(* CODESYS project Raspihats.library
   Description: Library for raspihats.com boards.
   Version: 1.0.0.0
   Title: Raspihats
   Author: Florin Costa
   DocFormat: reStructuredText
   Placeholder: Raspihats
   LanguageModelAttribute: qualified-access-only
   DefaultNamespace: Raspihats
   Company: Dabatop Industries SRL

Project tree, tasks and I/O mapping:
  libraries: Memory, 3.5.7.0 (3S - Smart Software Solutions GmbH); Raspberry Pi Peripherals, 3.5.13.0 (3S - Smart Software Solutions GmbH)
  I2CHAT/
    Globals/
      global variables I2CHAT_GVL
      data type I2CHAT_Command
      data type I2CHAT_ErrorCode
    Frame/
      function block I2CHAT_EncodeFrame [ST]
      function block I2CHAT_DecodeFrame [ST]
    Boards/
      function block I2CHAT_DI6acDQ6rly [ST]: AfterReadInputs, BeforeWriteOutputs
      function block I2CHAT_DI16ac [ST]: AfterReadInputs
      function block I2CHAT_DQ10rly [ST]: BeforeWriteOutputs
    I/O/
      function block I2CHAT_Transfer [ST]
      function block I2CHAT_DQ_Write [ST]
      function block I2CHAT_DI_Read [ST]
*)

// I2CHAT/Globals/I2CHAT_Command
{attribute 'qualified_only'}
{attribute 'strict'}
TYPE I2CHAT_Command :
(
    GET_BOARD_NAME                      := 16#10, 
    GET_FIRMWARE_VERSION                := 16#11, 
    GET_STATUS_WORD                     := 16#12, 
    RESET                               := 16#13,
 
    CWDT_SET_PERIOD                     := 16#14, 
    CWDT_GET_PERIOD                     := 16#15, 
    IRQ_GET_REG                         := 16#16, 
    IRQ_SET_REG                         := 16#17,  
 
    DI_GET_VALUE                        := 16#20, 
    DI_GET_CHANNEL_STATE                := 16#21, 
    DI_GET_COUNTER                      := 16#22, 
    DI_RESET_COUNTER                    := 16#23, 
    DI_RESET_ALL_COUNTERS               := 16#24, 
    DI_GET_COUNTERS_STATUS              := 16#25, 
    DI_GET_ENCODER                      := 16#26, 
    DI_RESET_ENCODER                    := 16#27, 
    DI_RESET_ALL_ENCODERS               := 16#28, 
    DI_GET_ENCODERS_STATUS              := 16#29, 
 
    DO_SET_POWER_ON_VALUE               := 16#30, 
    DO_GET_POWER_ON_VALUE               := 16#31, 
    DO_SET_SAFETY_VALUE                 := 16#32, 
    DO_GET_SAFETY_VALUE                 := 16#33, 
    DO_SET_VALUE                        := 16#34, 
    DO_GET_VALUE                        := 16#35, 
    DO_SET_CHANNEL_STATE                := 16#36, 
    DO_GET_CHANNEL_STATE                := 16#37
) USINT;
END_TYPE

// I2CHAT/Globals/I2CHAT_ErrorCode
{attribute 'qualified_only'}
{attribute 'strict'}
TYPE I2CHAT_ErrorCode :
(
	NO_ERROR := 0,
	I2C_WRITE_INCOMPLETE := 1,
	I2C_READ_INCOMPLETE := 2,
	BUFFER_OVERFLOW := 3,
	CRC_FAIL := 4,
	BAD_RESPONSE := 5
) UINT;
END_TYPE

// I2CHAT/Globals/I2CHAT_GVL
{attribute 'qualified_only'}
VAR_GLOBAL CONSTANT
	gc_uiFrameMinSize : UINT := 4; // 1(Id) + 1(Cmd) + 0(Payload) + 2(CRC16)
	gc_uiCrc16Size : UINT := 2;
END_VAR
VAR_GLOBAL
	g_usiFrameId : USINT := 0;
END_VAR

// I2CHAT/Boards/I2CHAT_DI6acDQ6rly
FUNCTION_BLOCK I2CHAT_DI6acDQ6rly EXTENDS i2c
VAR_INPUT
	udiDQValue : UDINT;
END_VAR
VAR_OUTPUT
	udiDIValue : UDINT;
	eErrorCode : I2CHAT_ErrorCode;
END_VAR
VAR
END_VAR

SUPER^();

CASE _iState OF
0:	
	IF SUPER^.init() THEN
		_iState := 10;
	END_IF	
	
END_CASE

METHOD AfterReadInputs : INT
VAR
	DI_Read : I2CHAT_DI_Read;
END_VAR
SUPER^.AfterReadInputs();

IF _iState = 10 THEN
	DI_Read(
		pI2CSlave := THIS
	);
	
	udiDIValue := DI_Read.udiValue;
	eErrorCode := DI_Read.eErrorCode;
END_IF
END_METHOD

METHOD BeforeWriteOutputs : INT
VAR
	DQ_Write : I2CHAT_DQ_Write;
	DI_Read: INT;
END_VAR
SUPER^.BeforeWriteOutputs();

IF _iState = 10 THEN
	DQ_Write(
		pI2CSlave := THIS, 
		udiValue := udiDQValue
	);
	
	eErrorCode := DQ_Write.eErrorCode;
END_IF
END_METHOD

END_FUNCTION_BLOCK

// I2CHAT/I/O/I2CHAT_DI_Read
FUNCTION_BLOCK I2CHAT_DI_Read
VAR_INPUT
	pI2CSlave : POINTER TO RasPi.i2c;
END_VAR
VAR_OUTPUT
	udiValue : UDINT;
	eErrorCode : I2CHAT_ErrorCode;
END_VAR
VAR
	ausiResponseData : ARRAY [0..3] OF USINT;
	Transfer : I2CHAT_Transfer;
END_VAR

Transfer(
	pI2CSlave := pI2CSlave,
	usiRequestCmd := I2CHAT_Command.DI_GET_VALUE,
	pusiRequestData := 0,
	uiRequestDataSize := 0,
	pusiResponseData := ADR(ausiResponseData),
	uiResponseDataSize := 4
);

IF Transfer.eErrorCode <> I2CHAT_ErrorCode.NO_ERROR THEN
	eErrorCode := Transfer.eErrorCode;
	RETURN;
END_IF

udiValue := ausiResponseData[0];
udiValue := udiValue + SHL(USINT_TO_UDINT(ausiResponseData[1]), 8);
udiValue := udiValue + SHL(USINT_TO_UDINT(ausiResponseData[2]), 16);
udiValue := udiValue + SHL(USINT_TO_UDINT(ausiResponseData[3]), 24);

END_FUNCTION_BLOCK

// I2CHAT/I/O/I2CHAT_Transfer
FUNCTION_BLOCK I2CHAT_Transfer
VAR_INPUT
	pI2CSlave : POINTER TO RasPi.i2c;
	usiRequestCmd : USINT;
	pusiRequestData : POINTER TO USINT;
	uiRequestDataSize : UINT;
	pusiResponseData : POINTER TO USINT;
	uiResponseDataSize : UINT;
END_VAR
VAR_OUTPUT
	eErrorCode : I2CHAT_ErrorCode;
END_VAR
VAR
	ausiBuffer : ARRAY [0..255] OF USINT;
	EncodeFrame : I2CHAT_EncodeFrame;
	DecodeFrame : I2CHAT_DecodeFrame;
	uiByteCnt : DINT;
END_VAR

eErrorCode := I2CHAT_ErrorCode.NO_ERROR;

I2CHAT_GVL.g_usiFrameId := (I2CHAT_GVL.g_usiFrameId + 1) AND 16#FF;

EncodeFrame(
	usiId := I2CHAT_GVL.g_usiFrameId,
	usiCmd := usiRequestCmd,
	pusiData := pusiRequestData,
	uiDataSize := uiRequestDataSize,
	pusiBuffer := ADR(ausiBuffer),
	uiBufferSize := SIZEOF(ausiBuffer)
);

IF EncodeFrame.eErrorCode <> I2CHAT_ErrorCode.NO_ERROR THEN
	eErrorCode := EncodeFrame.eErrorCode;
	RETURN;
END_IF

// Write I2C-HAT request
uiByteCnt := pI2CSlave^.write(ADR(ausiBuffer), EncodeFrame.uiEncodeSize);
IF uiByteCnt <> EncodeFrame.uiEncodeSize THEN
	eErrorCode := I2CHAT_ErrorCode.I2C_WRITE_INCOMPLETE;
	RETURN;
END_IF

// Read I2C-HAT response
uiByteCnt:= pI2CSlave^.read(ADR(ausiBuffer), I2CHAT_GVL.gc_uiFrameMinSize + uiResponseDataSize);
IF uiByteCnt <> (I2CHAT_GVL.gc_uiFrameMinSize + uiResponseDataSize) THEN
	eErrorCode := I2CHAT_ErrorCode.I2C_READ_INCOMPLETE;
	RETURN;
END_IF

DecodeFrame(
	pusiBuffer := ADR(ausiBuffer),
	uiBufferSize := I2CHAT_GVL.gc_uiFrameMinSize + uiResponseDataSize,
	pusiData := pusiResponseData,
	uiDataSize := uiResponseDataSize
);

IF DecodeFrame.eErrorCode <> I2CHAT_ErrorCode.NO_ERROR THEN
	eErrorCode := DecodeFrame.eErrorCode;
	RETURN;
END_IF

IF DecodeFrame.usiId <> EncodeFrame.usiId OR DecodeFrame.usiCmd <> EncodeFrame.usiCmd THEN
	eErrorCode := I2CHAT_ErrorCode.BAD_RESPONSE;
END_IF

END_FUNCTION_BLOCK

// I2CHAT/Frame/I2CHAT_EncodeFrame
FUNCTION_BLOCK I2CHAT_EncodeFrame
VAR_INPUT
	// input frame
	usiId : USINT;
	usiCmd : USINT;
	pusiData : POINTER TO USINT;
	uiDataSize : UINT;
	// encode buffer
	pusiBuffer : POINTER TO USINT;
	uiBufferSize : UINT;
END_VAR
VAR_OUTPUT
	uiEncodeSize : UINT;
	eErrorCode : I2CHAT_ErrorCode;
END_VAR
VAR
	uiEncodeIndex : UINT;
	uiIndex : UINT;
	uiCrc16 : UINT;
END_VAR

IF (I2CHAT_GVL.gc_uiFrameMinSize + uiDataSize) <= uiBufferSize THEN
	uiEncodeIndex := 0;
	
	pusiBuffer[uiEncodeIndex] := usiId;
	uiEncodeIndex := uiEncodeIndex + 1;
    
	pusiBuffer[uiEncodeIndex] := usiCmd;
	uiEncodeIndex := uiEncodeIndex + 1;

	IF uiDataSize > 0 THEN
		FOR uiIndex := 0 TO uiDataSize - 1 DO
			pusiBuffer[uiEncodeIndex] := pusiData[uiIndex];
			uiEncodeIndex := uiEncodeIndex + 1;		
		END_FOR
	END_IF

	uiCrc16 := MEM.CRC16_Modbus(pMemoryBlock := pusiBuffer, uiLength := uiEncodeIndex);

	pusiBuffer[uiEncodeIndex] := UINT_TO_USINT(uiCrc16);
	uiEncodeIndex := uiEncodeIndex + 1;
	
	pusiBuffer[uiEncodeIndex] := UINT_TO_USINT(SHR(uiCrc16, 8));
	uiEncodeIndex := uiEncodeIndex + 1;	
	
	uiEncodeSize := uiEncodeIndex;
	eErrorCode := I2CHAT_ErrorCode.NO_ERROR;
ELSE 
	uiEncodeSize := 0;	// Nothing Encoded
	eErrorCode := I2CHAT_ErrorCode.BUFFER_OVERFLOW;
END_IF

END_FUNCTION_BLOCK

// I2CHAT/Frame/I2CHAT_DecodeFrame
FUNCTION_BLOCK I2CHAT_DecodeFrame
VAR_INPUT
	// decode buffer
	pusiBuffer : POINTER TO USINT;
	uiBufferSize : UINT;
	// frame payload buffer
	pusiData : POINTER TO USINT;
	uiDataSize : UINT;
END_VAR
VAR_OUTPUT
	usiId : USINT;
	usiCmd : USINT;
	uiDecodeSize : UINT;
	eErrorCode : I2CHAT_ErrorCode;
END_VAR
VAR
	uiDecodeIndex : UINT;
	uiIndex : UINT;
	uiCrc16 : UINT;
END_VAR

IF uiBufferSize >= I2CHAT_GVL.gc_uiFrameMinSize AND uiDataSize >= (uiBufferSize - I2CHAT_GVL.gc_uiFrameMinSize) THEN
	uiDecodeIndex := 0;
	
	usiId := pusiBuffer[uiDecodeIndex]; 
	uiDecodeIndex := uiDecodeIndex + 1;
    
	usiCmd := pusiBuffer[uiDecodeIndex]; 
	uiDecodeIndex := uiDecodeIndex + 1;

	uiDataSize := uiBufferSize - I2CHAT_GVL.gc_uiFrameMinSize;
	IF uiDataSize > 0 THEN
		FOR uiIndex := 0 TO uiDataSize - 1 DO
			pusiData[uiIndex] := pusiBuffer[uiDecodeIndex];
			uiDecodeIndex := uiDecodeIndex + 1;	
		END_FOR
	END_IF

	uiCrc16 := USINT_TO_UINT(pusiBuffer[uiDecodeIndex]); 
	uiDecodeIndex := uiDecodeIndex + 1;
	
	uiCrc16 := uiCrc16 + SHL(USINT_TO_UINT(pusiBuffer[uiDecodeIndex]), 8); 
	uiDecodeIndex := uiDecodeIndex + 1;
	
	IF MEM.CRC16_Modbus(pMemoryBlock := pusiBuffer, uiLength := uiDecodeIndex - I2CHAT_GVL.gc_uiCrc16Size) = uiCrc16 THEN
		uiDecodeSize := uiDecodeIndex;
		eErrorCode := I2CHAT_ErrorCode.NO_ERROR;
	ELSE
		uiDecodeSize := 0;	
		eErrorCode := I2CHAT_ErrorCode.CRC_FAIL;
	END_IF
ELSE 
	uiDecodeSize := 0;
	eErrorCode := I2CHAT_ErrorCode.BUFFER_OVERFLOW;
END_IF

END_FUNCTION_BLOCK

// I2CHAT/I/O/I2CHAT_DQ_Write
FUNCTION_BLOCK I2CHAT_DQ_Write
VAR_INPUT
	pI2CSlave : POINTER TO RasPi.i2c;
	udiValue : UDINT;
END_VAR
VAR_OUTPUT
	eErrorCode : I2CHAT_ErrorCode;
END_VAR
VAR
	ausiRequestData : ARRAY [0..3] OF USINT;
	ausiResponseData : ARRAY [0..3] OF USINT;
	Transfer : I2CHAT_Transfer;
END_VAR

ausiRequestData[0] := UDINT_TO_USINT(udiValue);
ausiRequestData[1] := UDINT_TO_USINT(SHR(udiValue, 8));
ausiRequestData[2] := UDINT_TO_USINT(SHR(udiValue, 16));
ausiRequestData[3] := UDINT_TO_USINT(SHR(udiValue, 24));

Transfer(
	pI2CSlave := pI2CSlave,
	usiRequestCmd := I2CHAT_Command.DO_SET_VALUE,
	pusiRequestData := ADR(ausiRequestData),
	uiRequestDataSize := 4,
	pusiResponseData := ADR(ausiResponseData),
	uiResponseDataSize := 4
);

IF Transfer.eErrorCode <> I2CHAT_ErrorCode.NO_ERROR THEN
	eErrorCode := Transfer.eErrorCode;
	RETURN;
END_IF

//Check that response frame data is identical to request frame data
IF MEM.Compare(ADR(ausiRequestData), ADR(ausiResponseData), 4) <> 0 THEN
	eErrorCode := I2CHAT_ErrorCode.BAD_RESPONSE;
ELSE
	eErrorCode := I2CHAT_ErrorCode.NO_ERROR;
END_IF

END_FUNCTION_BLOCK

// I2CHAT/Boards/I2CHAT_DI16ac
FUNCTION_BLOCK I2CHAT_DI16ac EXTENDS i2c
VAR_OUTPUT
	udiDIValue : UDINT;
	eErrorCode : I2CHAT_ErrorCode;
END_VAR
VAR
END_VAR

SUPER^();

CASE _iState OF
0:	
	IF SUPER^.init() THEN
		_iState := 10;
	END_IF	
	
END_CASE

METHOD AfterReadInputs : INT
VAR
	DI_Read : I2CHAT_DI_Read;
END_VAR
SUPER^.AfterReadInputs();

IF _iState = 10 THEN
	DI_Read(
		pI2CSlave := THIS
	);
	
	udiDIValue := DI_Read.udiValue;
	eErrorCode := DI_Read.eErrorCode;
END_IF
END_METHOD

END_FUNCTION_BLOCK

// I2CHAT/Boards/I2CHAT_DQ10rly
FUNCTION_BLOCK I2CHAT_DQ10rly EXTENDS i2c
VAR_INPUT
	udiDQValue : UDINT;
END_VAR
VAR_OUTPUT
	eErrorCode : I2CHAT_ErrorCode;
END_VAR
VAR
END_VAR

SUPER^();

CASE _iState OF
0:	
	IF SUPER^.init() THEN
		_iState := 10;
	END_IF	
	
END_CASE

METHOD BeforeWriteOutputs : INT
VAR
	DQ_Write : I2CHAT_DQ_Write;
	DI_Read: INT;
END_VAR
SUPER^.BeforeWriteOutputs();

IF _iState = 10 THEN
	DQ_Write(
		pI2CSlave := THIS, 
		udiValue := udiDQValue
	);
	
	eErrorCode := DQ_Write.eErrorCode;
END_IF
END_METHOD

END_FUNCTION_BLOCK
